(* CODESYS project EDS_V2_neu.project

Project tree, tasks and I/O mapping:
  CODESYS_SoftMotion_Win_V3 : CODESYS SoftMotion Win V3, 3S - Smart Software Solutions GmbH, order no. 309021, version 3.5.10.20
    application Application
      libraries: crane-control-lib, 1.0.3 (TUD)
      task VISU_TASK (cyclic, interval 100 ms, priority 31) calls VisuElems.Visu_Prg
      task Task (cyclic, interval t#20ms, priority 1) calls Motion_PRG_Motion, Motion_PRG_Control
      visualisation Visualization
      function block Bandsteuerung [SFC]: Init_active, Gleiten_active, Brems_active
      global variables GVL
      function Vmax [ST]
      program Motion_PRG_Control [FBD]
      program Motion_PRG_Motion [FBD]
      function block Kransteuerung [SFC]: brems_aufw_active, beschl_abw_active, Ruhelage_active
    SoftMotion General Axis Pool
      VA1_Band : SM_Drive_Virtual, 3S - Smart Software Solutions GmbH, order no. 1805, version 4.0.0.0
          settings: wDriveID = 0; iMovementType = 0
      VA2_Kran : SM_Drive_Virtual, 3S - Smart Software Solutions GmbH, order no. 1805, version 4.0.0.0
  libraries: VisuSymbols, 3.5.10.0 (System)
  text list GlobalTextList
*)

// CODESYS_SoftMotion_Win_V3/Application/GVL
VAR_GLOBAL
	
	jerk:REAL := 0; //unendlicher Ruck für geschwindigkeitsoptimale Steuerung
(* Steuervariablen (werden durch die Visualisierung gesetzt) *)
	Anlage_Ein:BOOL:=FALSE; (* Steuervariable zum Ein- und Ausschalten der Anlage *)
	Erzeuge_Paket_schwarz:BOOL; (* Es soll ein neues schwarzes Paket erzeugt werden *)
	Erzeuge_Paket_rot:BOOL; (* Es soll ein neues rotes Paket erzeugt werden *)
	
	(* Achsbezogene Variablen (repraesentieren aktuelle Messwerte der Achsen) *)
	Vact_Foerderbandachse:REAL; (* Aktuelle Winkelgeschwindigkeit der Foerderbandachse (in Grad/s) *)
	Vact_Foerderband:REAL; (* Aktuelle Geschwindigkeit des Foerderbandes (in mm/s) *)
	Vact_Kran1:REAL; (* Aktuelle vertikale Geschwindigkeit von Kran 1 (in mm/s) *)
	Posact_Kran1:REAL; (* Aktuelle vertikale Position von Kran 1 (in mm) *)
	
	(* Sensoren (werden durch den Simulator gesetzt) *)
	Messwert_Farbsensor:INT; (* Aktueller Messwert des Farbsensors (0=kein Paket; CONST.SCHWARZ=schwarzes Paket; CONST.ROT=rotes Paket) *)
	Kran1_In_Startpos:BOOL; (* Kran 1 befindet sich in seiner Startposition *)
	Kran1_In_Greifpos:BOOL; (* Kran 1 befindet sich in seiner Greifposition *)
	A_Band:REAL:=100;//*CONST.PI/180*RADIUS_FOERDERBANDACHSE; //Förderbeschleunigung Band in mm/s^2 //in Grad/s^2
	V_Band:REAL:=50;//*CONST.PI/180*RADIUS_FOERDERBANDACHSE ;//in mm/s //in Grad/s
	
	deltaT:REAL:=(GREIFPOS_X_KRAN1-POS_X_SENSOR)/(V_Band);(* berechnete Zeit des Paketes von Sensor zu Kran = Bewegungszeit des Krans in eine Richtung = 11.37s*)
	
END_VAR

// CODESYS_SoftMotion_Win_V3/Application/Motion_PRG_Motion
PROGRAM Motion_PRG_Motion
VAR_OUTPUT
	br_PowerVA1: BOOL;
	bd_PowerVA1: BOOL;
	bu_PowerVA1: BOOL;
	er_PowerVA1: BOOL;
	ID_PowerVA1: SMC_ERROR;
	st_PowerVA1: BOOL;
	
	don_accVA1: BOOL;
	bu_accVA1: BOOL;
	ab_accVA1: BOOL;
	er_accVA1: BOOL;
	ID_accVA1: SMC_ERROR;
	
	inVelocity_glVA1: BOOL;
	bu_glVA1: BOOL;
	ab_glVA1: BOOL;
	er_glVA1: BOOL;
	ID_glVA1: SMC_ERROR;
	
	don_decVA1: BOOL;
	bu_decVA1: BOOL;
	er_decVA1: BOOL;
	ID_decVA1: SMC_ERROR;
	
	
	st_PowerVA2: BOOL;
	bd_PowerVA2: BOOL;
	bu_PowerVA2: BOOL;
	br_PowerVA2: BOOL;
	er_PowerVA2: BOOL;
	ID_PowerVA2: SMC_ERROR;
	
	don_accVA2: BOOL;
	bu_accVA2: BOOL;
	er_accVA2: BOOL;
	ab_accVA2: BOOL;
	ID_accVA2: SMC_ERROR;
	
	inVelocity_glVA2: BOOL;
	bu_glVA2: BOOL;
	ab_glVA2: BOOL;
	ID_glVA2: SMC_ERROR;
	er_glVA2: BOOL;
	
	don_decVA2: BOOL;
	bu_decVA2: BOOL;
	er_decVA2: BOOL;
	ID_decVA2: SMC_ERROR;
	
END_VAR

VAR
	Power_VA1: MC_Power;
	Power_VA2: MC_Power;
	MC_Stop_Kran: MC_Stop;
	MC_MoveAbsolute_Kran: MC_MoveAbsolute;
	MC_MoveVelocity_Kran: MC_MoveVelocity;
	MC_MoveVelocity_Band :MC_MoveVelocity;
	MC_MoveAbsolute_Band: MC_MoveAbsolute;
	MC_Stop_Band: MC_Stop;
	
	
	
	don_reset: BOOL;
	bu_reset: BOOL;
	er_reset: BOOL;
	ID_reset: SMC_ERROR;
	MC_Reset_Band: MC_Reset;
	MC_Reset_Kran: MC_Reset;
END_VAR

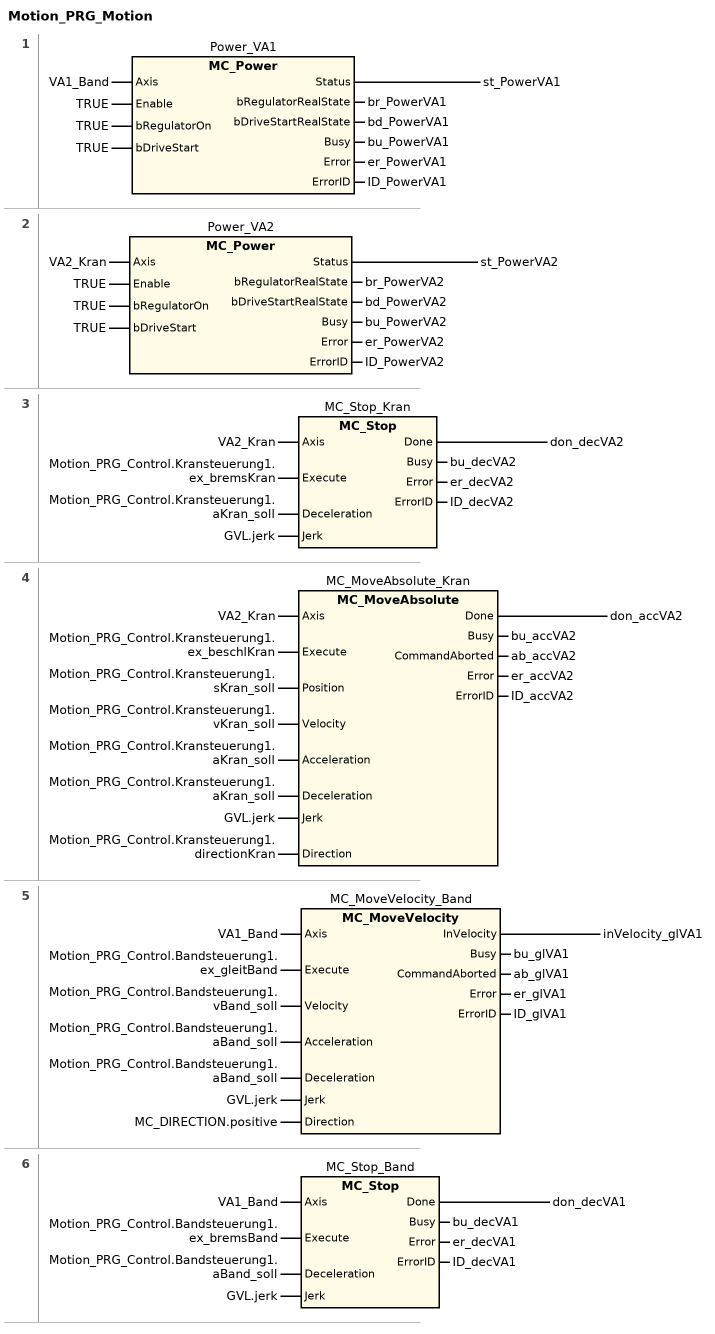
// NETWORK 1
Power_VA1(
    Axis := VA1_Band,
    Enable := TRUE,
    bRegulatorOn := TRUE,
    bDriveStart := TRUE,
    bRegulatorRealState => br_PowerVA1,
    bDriveStartRealState => bd_PowerVA1,
    Busy => bu_PowerVA1,
    Error => er_PowerVA1,
    ErrorID => ID_PowerVA1); // MC_Power
st_PowerVA1 := Power_VA1.Status;

// NETWORK 2
Power_VA2(
    Axis := VA2_Kran,
    Enable := TRUE,
    bRegulatorOn := TRUE,
    bDriveStart := TRUE,
    bRegulatorRealState => br_PowerVA2,
    bDriveStartRealState => bd_PowerVA2,
    Busy => bu_PowerVA2,
    Error => er_PowerVA2,
    ErrorID => ID_PowerVA2); // MC_Power
st_PowerVA2 := Power_VA2.Status;

// NETWORK 3
MC_Stop_Kran(
    Axis := VA2_Kran,
    Execute := Motion_PRG_Control.Kransteuerung1.ex_bremsKran,
    Deceleration := Motion_PRG_Control.Kransteuerung1.aKran_soll,
    Jerk := GVL.jerk,
    Busy => bu_decVA2,
    Error => er_decVA2,
    ErrorID => ID_decVA2); // MC_Stop
don_decVA2 := MC_Stop_Kran.Done;

// NETWORK 4
MC_MoveAbsolute_Kran(
    Axis := VA2_Kran,
    Execute := Motion_PRG_Control.Kransteuerung1.ex_beschlKran,
    Position := Motion_PRG_Control.Kransteuerung1.sKran_soll,
    Velocity := Motion_PRG_Control.Kransteuerung1.vKran_soll,
    Acceleration := Motion_PRG_Control.Kransteuerung1.aKran_soll,
    Deceleration := Motion_PRG_Control.Kransteuerung1.aKran_soll,
    Jerk := GVL.jerk,
    Direction := Motion_PRG_Control.Kransteuerung1.directionKran,
    Busy => bu_accVA2,
    CommandAborted => ab_accVA2,
    Error => er_accVA2,
    ErrorID => ID_accVA2); // MC_MoveAbsolute
don_accVA2 := MC_MoveAbsolute_Kran.Done;

// NETWORK 5
MC_MoveVelocity_Band(
    Axis := VA1_Band,
    Execute := Motion_PRG_Control.Bandsteuerung1.ex_gleitBand,
    Velocity := Motion_PRG_Control.Bandsteuerung1.vBand_soll,
    Acceleration := Motion_PRG_Control.Bandsteuerung1.aBand_soll,
    Deceleration := Motion_PRG_Control.Bandsteuerung1.aBand_soll,
    Jerk := GVL.jerk,
    Direction := MC_DIRECTION.positive,
    Busy => bu_glVA1,
    CommandAborted => ab_glVA1,
    Error => er_glVA1,
    ErrorID => ID_glVA1); // MC_MoveVelocity
inVelocity_glVA1 := MC_MoveVelocity_Band.InVelocity;

// NETWORK 6
MC_Stop_Band(
    Axis := VA1_Band,
    Execute := Motion_PRG_Control.Bandsteuerung1.ex_bremsBand,
    Deceleration := Motion_PRG_Control.Bandsteuerung1.aBand_soll,
    Jerk := GVL.jerk,
    Busy => bu_decVA1,
    Error => er_decVA1,
    ErrorID => ID_decVA1); // MC_Stop
don_decVA1 := MC_Stop_Band.Done;

END_PROGRAM

// CODESYS_SoftMotion_Win_V3/Application/Motion_PRG_Control
PROGRAM Motion_PRG_Control
VAR
	Simulator1:Simulator; (* Foerderbandsimulator aus der 'crane-control-lib' *)
	
	
	Kransteuerung1: Kransteuerung;
	Bandsteuerung1: Bandsteuerung;

	
	
END_VAR

VAR_OUTPUT
	
	ex_gleitBand: BOOL;
	ex_bremsBand: BOOL;
	ex_beschlKran: BOOL;
	ex_gleitKran: BOOL;
	ex_bremsKran:BOOL;
	aKran_soll:LREAL;
	vKran_soll:LREAL; //Sollwert der vertikalen Geschwindigkeit des Krans in mm/s
	sKran_soll:LREAL; //Sollwert des vertikalen Weges des Krans in mm 
	vBand_soll: LREAL;
	aBand_soll:LREAL;		
	ex_beschlBand: BOOL;
END_VAR

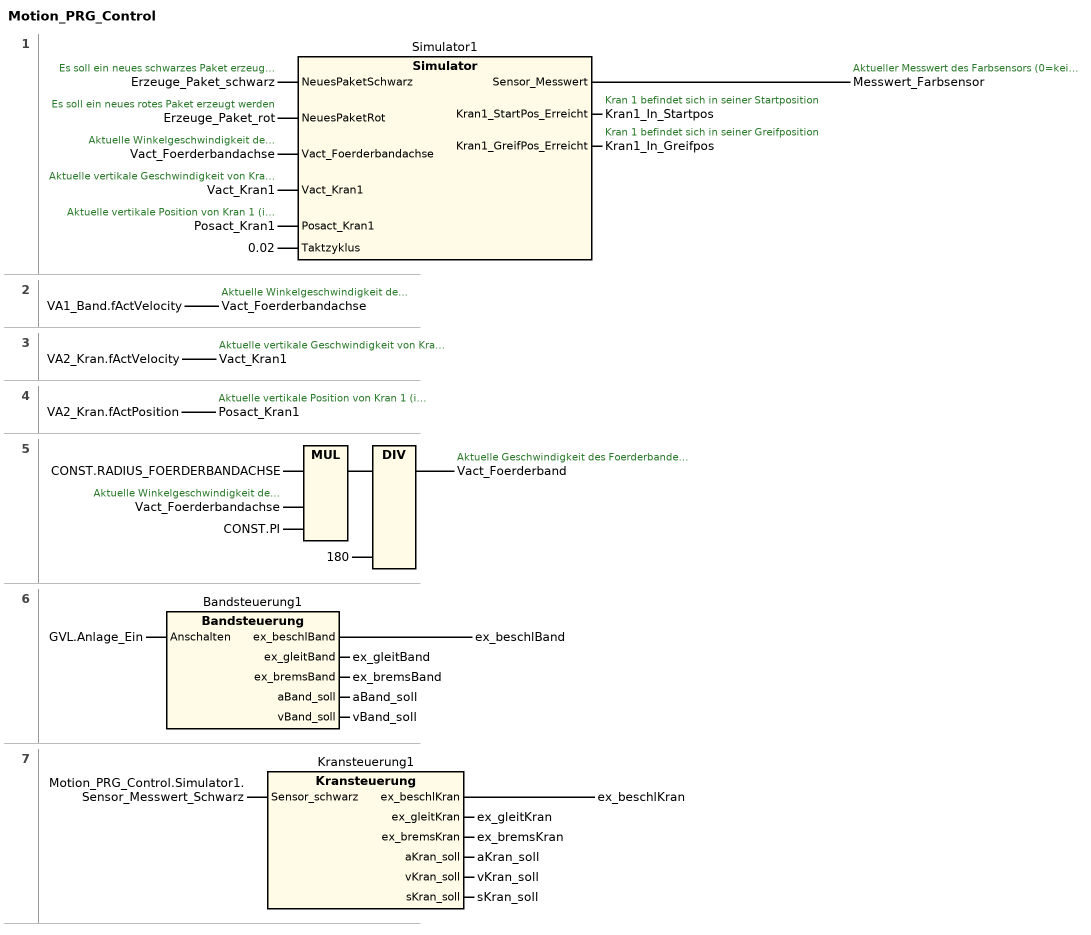
// NETWORK 1
//   Simulator1: Foerderbandsimulator aus der 'crane-control-lib'
//   Erzeuge_Paket_schwarz: Es soll ein neues schwarzes Paket erzeugt werden
//   Erzeuge_Paket_rot: Es soll ein neues rotes Paket erzeugt werden
//   Vact_Foerderbandachse: Aktuelle Winkelgeschwindigkeit der Foerderbandachse (in Grad/s)
//   Vact_Kran1: Aktuelle vertikale Geschwindigkeit von Kran 1 (in mm/s)
//   Posact_Kran1: Aktuelle vertikale Position von Kran 1 (in mm)
//   Kran1_In_Startpos: Kran 1 befindet sich in seiner Startposition
//   Kran1_In_Greifpos: Kran 1 befindet sich in seiner Greifposition
//   Messwert_Farbsensor: Aktueller Messwert des Farbsensors (0=kein Paket; CONST.SCHWARZ=schwarzes Paket; CONST.ROT=rotes Paket)
Simulator1(
    NeuesPaketSchwarz := Erzeuge_Paket_schwarz,
    NeuesPaketRot := Erzeuge_Paket_rot,
    Vact_Foerderbandachse := Vact_Foerderbandachse,
    Vact_Kran1 := Vact_Kran1,
    Posact_Kran1 := Posact_Kran1,
    Taktzyklus := 0.02,
    Kran1_StartPos_Erreicht => Kran1_In_Startpos,
    Kran1_GreifPos_Erreicht => Kran1_In_Greifpos); // Simulator
Messwert_Farbsensor := Simulator1.Sensor_Messwert;

// NETWORK 2
//   Vact_Foerderbandachse: Aktuelle Winkelgeschwindigkeit der Foerderbandachse (in Grad/s)
Vact_Foerderbandachse := VA1_Band.fActVelocity;

// NETWORK 3
//   Vact_Kran1: Aktuelle vertikale Geschwindigkeit von Kran 1 (in mm/s)
Vact_Kran1 := VA2_Kran.fActVelocity;

// NETWORK 4
//   Posact_Kran1: Aktuelle vertikale Position von Kran 1 (in mm)
Posact_Kran1 := VA2_Kran.fActPosition;

// NETWORK 5
//   Vact_Foerderbandachse: Aktuelle Winkelgeschwindigkeit der Foerderbandachse (in Grad/s)
//   Vact_Foerderband: Aktuelle Geschwindigkeit des Foerderbandes (in mm/s)
Vact_Foerderband := (CONST.RADIUS_FOERDERBANDACHSE * Vact_Foerderbandachse * CONST.PI) / 180;

// NETWORK 6
Bandsteuerung1(
    Anschalten := GVL.Anlage_Ein,
    ex_gleitBand => ex_gleitBand,
    ex_bremsBand => ex_bremsBand,
    aBand_soll => aBand_soll,
    vBand_soll => vBand_soll); // Bandsteuerung
ex_beschlBand := Bandsteuerung1.ex_beschlBand;

// NETWORK 7
Kransteuerung1(
    Sensor_schwarz := Motion_PRG_Control.Simulator1.Sensor_Messwert_Schwarz,
    ex_gleitKran => ex_gleitKran,
    ex_bremsKran => ex_bremsKran,
    aKran_soll => aKran_soll,
    vKran_soll => vKran_soll,
    sKran_soll => sKran_soll); // Kransteuerung
ex_beschlKran := Kransteuerung1.ex_beschlKran;

END_PROGRAM

// CODESYS_SoftMotion_Win_V3/Application/Bandsteuerung
FUNCTION_BLOCK Bandsteuerung


VAR
	TAU1 :TIME :=REAL_TO_TIME(V_Band/A_Band*10000);
	T1: BOOL:=FALSE;
	T2: BOOL:=FALSE;
END_VAR

VAR_OUTPUT
	ex_resetBand:BOOL:=FALSE;
	ex_beschlBand: BOOL:=FALSE;
	ex_gleitBand: BOOL:=FALSE;
	ex_bremsBand: BOOL:=FALSE;
	aBand_soll: LREAL;
	vBand_soll: LREAL;
	sBand_soll: LREAL;
END_VAR

VAR_INPUT
	Anschalten:BOOL:=GVL.Anlage_Ein;
END_VAR

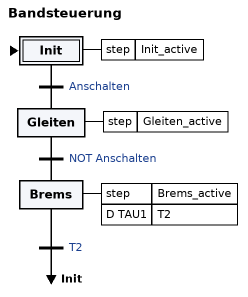
INITIAL_STEP Init:
    Init_active(N);  // step action
END_STEP
TRANSITION FROM Init TO Gleiten
    := Anschalten;
END_TRANSITION
STEP Gleiten:
    Gleiten_active(N);  // step action
END_STEP
TRANSITION FROM Gleiten TO Brems
    := NOT Anschalten;
END_TRANSITION
STEP Brems:
    Brems_active(N);  // step action
    T2(D, TAU1);
END_STEP
TRANSITION FROM Brems TO Init
    := T2;
END_TRANSITION

ACTION Init_active:

END_ACTION

ACTION Gleiten_active:
ex_beschlBand:=FALSE;
ex_gleitBand:=TRUE;
ex_bremsBand:=FALSE;
aBand_soll:=GVL.A_Band;
vBand_soll:=GVL.V_Band ;
END_ACTION

ACTION Brems_active:

ex_beschlBand:=FALSE;
ex_gleitBand:=FALSE;
ex_bremsBand:=TRUE;
aBand_soll:=A_Band;
vBand_soll:=0 ;
END_ACTION

END_FUNCTION_BLOCK

// CODESYS_SoftMotion_Win_V3/Application/Kransteuerung
FUNCTION_BLOCK Kransteuerung
VAR_INPUT
	Sensor_schwarz: BOOL := FALSE;
END_VAR

VAR_OUTPUT
	ex_resetKran:BOOL:=FALSE;
	directionKran:MC_DIRECTION;
	ex_beschlKran:BOOL;
	ex_gleitKran:BOOL;
	ex_bremsKran:BOOL;
	aKran_soll:LREAL;
	vKran_soll:LREAL; //Sollwert der vertikalen Geschwindigkeit des Krans in mm/s
	sKran_soll:LREAL; //Sollwert des vertikalen Weges des Krans in mm 
END_VAR

VAR
	deltaS:LREAL := CONST.GREIFPOS_Y_KRAN-CONST.STARTPOS_Y_KRAN;
	V_max:LREAL:= Vmax(deltaS,GVL.deltaT,CONST.A_MAX);
	TAU1:TIME := LREAL_TO_TIME(V_max/CONST.A_MAX*1000) ;
	TAU2:TIME := LREAL_TO_TIME((deltaS/V_max-V_max/CONST.A_MAX)*1000);
	TAU3:TIME := TAU1;
	t0: BOOL := FALSE;
	t1: BOOL := FALSE;
	t2: BOOL := FALSE;
	t3: BOOL := FALSE;
	t4: BOOL := FALSE;
	t5: BOOL := FALSE;
	t6: BOOL := FALSE;
	
	
	
END_VAR

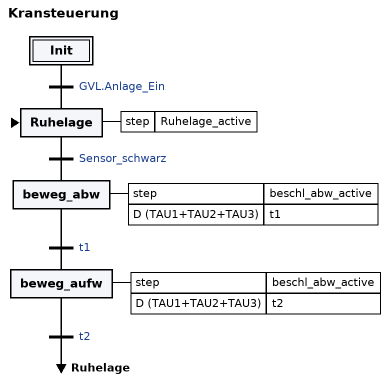
INITIAL_STEP Init:
END_STEP
TRANSITION FROM Init TO Ruhelage
    := GVL.Anlage_Ein;
END_TRANSITION
STEP Ruhelage:
    Ruhelage_active(N);  // step action
END_STEP
TRANSITION FROM Ruhelage TO beweg_abw
    := Sensor_schwarz;
END_TRANSITION
STEP beweg_abw:
    beschl_abw_active(N);  // step action
    t1(D, (TAU1+TAU2+TAU3));
END_STEP
TRANSITION FROM beweg_abw TO beweg_aufw
    := t1;
END_TRANSITION
STEP beweg_aufw:
    beschl_abw_active(N);  // step action
    t2(D, (TAU1+TAU2+TAU3));
END_STEP
TRANSITION FROM beweg_aufw TO Ruhelage
    := t2;
END_TRANSITION

ACTION brems_aufw_active:
ex_resetKran:=TRUE;
END_ACTION

ACTION beschl_abw_active:
ex_beschlKran:=TRUE;
ex_gleitKran:=FALSE;
ex_bremsKran:=FALSE;
aKran_soll:=CONST.A_MAX;
vKran_soll:=V_max;
sKran_soll:=CONST.STARTPOS_Y_KRAN;
directionKran:= MC_DIRECTION.negative;
END_ACTION

ACTION Ruhelage_active:
ex_beschlKran:=FALSE;
ex_gleitKran:=FALSE;
ex_bremsKran:=TRUE;

sKran_soll:=CONST.STARTPOS_Y_KRAN;
END_ACTION

END_FUNCTION_BLOCK

// CODESYS_SoftMotion_Win_V3/Application/Vmax
FUNCTION Vmax : LREAL
VAR_INPUT
	deltaS:LREAL;
	deltaT:LREAL;
	aMax:LREAL;
END_VAR
VAR
END_VAR

Vmax := deltaT*aMax/2*(1-SQRT(1-4*deltaS*aMax/EXPT(deltaT*aMax,2)));

END_FUNCTION

// CODESYS_SoftMotion_Win_V3/Application/Visualization
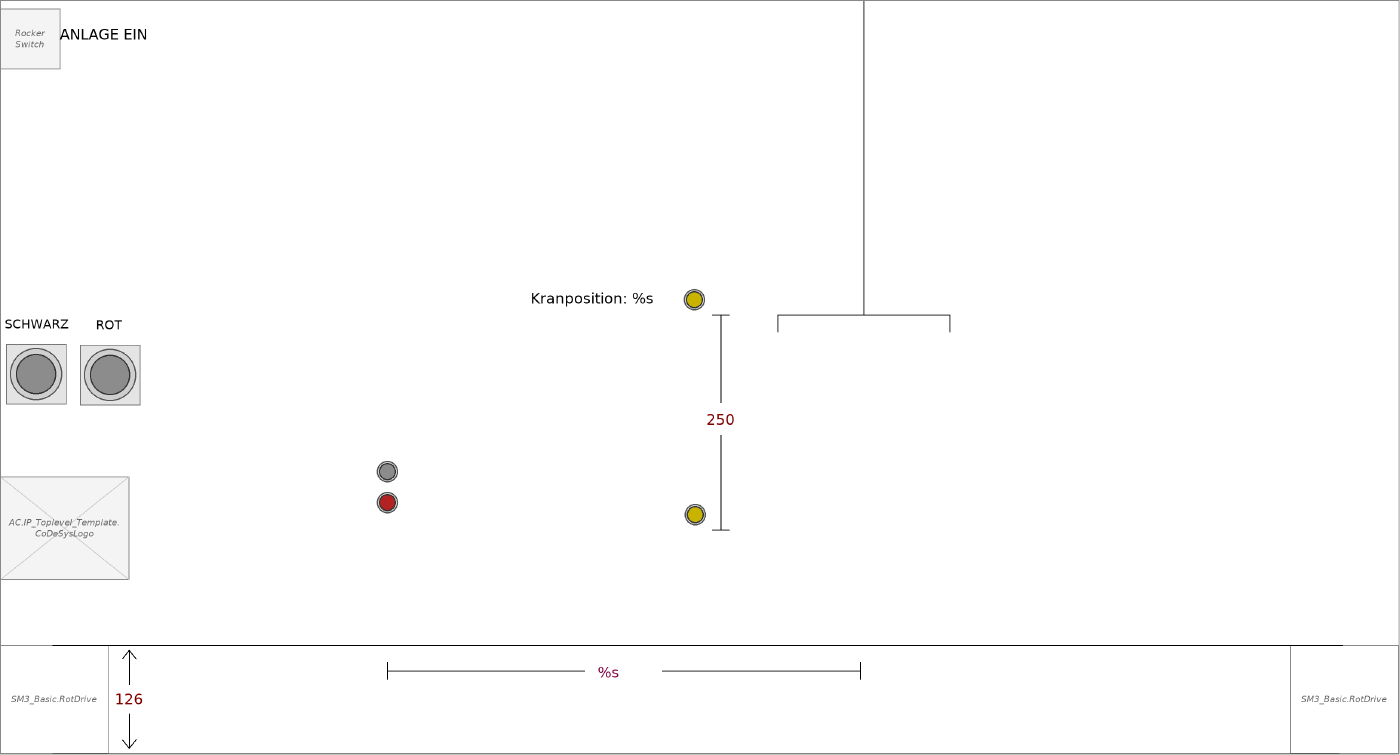
VISUALIZATION Visualization  // 1628x878
    Group (615,-2 490x619)
        p3560616238: GREIFPOS_X_KRAN1-925
        Line (389,0) (389,360)
        Line (389,50) (389,368)
            p2738717112: VA2_Kran.fActPosition
        Line (289,368) (489,368)
            p2738717112: VA2_Kran.fActPosition
        Line (489,368) (489,388)
            p2738717112: VA2_Kran.fActPosition
        Line (289,368) (289,388)
            p2738717112: VA2_Kran.fActPosition
        Textfield (117,334 60x30), "%s", text variable: Posact_Kran1
        Lamp1 (178,586 31x29), variable: Motion_PRG_Control.Simulator1.Kran1_GreifPos_Erreicht, style: Lamp-Lamp1-Yellow
        Lamp1 (177,336 31x29), variable: Motion_PRG_Control.Simulator1.Kran1_StartPos_Erreicht, style: Lamp-Lamp1-Yellow
        Line (223,368) (223,470)
        Line (223,508) (223,618)
        Label (189,473 68x34), "250"
        Line (213,618) (233,618)
        Line (213,368) (233,368)
        Label (0,334 117x30), "Kranposition:"
    Frame (0,750 126x126)
        shows SM3_Basic.RotDrive(m_Input_AXISREF := VA1_Band)
    Frame (1500,750 126x126)
        shows SM3_Basic.RotDrive(m_Input_AXISREF := VA1_Band)
        p3560616238: LAENGE_FOERDERBAND-1500
    Line (0,0) (1626,0)
    RockerSwitch (0,10 70x70), variable: GVL.Anlage_Ein, behaviour: TOGGLE, style: Switch-RockerSwitch-Gray
    Image (0,554 150x120), colour toggle: INT_TO_BOOL(Motion_PRG_Control.Simulator1.Paket1_Farbe - 1), invisible if: Motion_PRG_Control.Simulator1.Paket1_Unsichtbar, image: AC.IP_Toplevel_Template.CoDeSysLogo
        p3560616238: Motion_PRG_Control.Simulator1.Paket1_Pos_x
        p2738717112: Motion_PRG_Control.Simulator1.Paket1_Pos_y
    PushSwitch (7,400 70x70), variable: Erzeuge_Paket_schwarz, behaviour: TAP, style: Switch-PushSwitch-Gray
    Image (0,554 150x120), colour toggle: INT_TO_BOOL(Motion_PRG_Control.Simulator1.Paket2_Farbe - 1), invisible if: Motion_PRG_Control.Simulator1.Paket2_Unsichtbar, image: AC.IP_Toplevel_Template.CoDeSysLogo
        p3560616238: Motion_PRG_Control.Simulator1.Paket2_Pos_x
        p2738717112: Motion_PRG_Control.Simulator1.Paket2_Pos_y
    Line (61,750) (1061,750)
    Line (61,876) (1061,876)
    Label (0,360 86x34), "SCHWARZ"
    Label (56,23 129x34), "ANLAGE EIN"
    Lamp1 (435,534 31x29), variable: Motion_PRG_Control.Simulator1.Sensor_Messwert_Schwarz, style: Lamp-Lamp1-Gray
    Line (450,780) (650,780)
    Line (450,770) (450,790)
    Line (1000,770) (1000,790)
        p3560616238: GREIFPOS_X_KRAN1-925
    Line (770,780) (970,780)
        p3560616238: (GREIFPOS_X_KRAN1-925)/2
    Line (364,317)
    Line (150,756) (150,796)
    Line (150,830) (150,870)
    Label (116,796 68x34), "126"
    Line (150,756) (158,766)
    Line (150,756) (142,766)
    Line (142,860) (150,870)
    Line (158,860) (150,870)
    Line (561,750) (1561,750)
        p3560616238: LAENGE_FOERDERBAND-1500
    Line (557,876) (1557,876)
        p3560616238: LAENGE_FOERDERBAND-1500
    Line (480,780) (680,780)
        p3560616238: (GREIFPOS_X_KRAN1-925)/2
    Line (800,780) (1000,780)
        p3560616238: (GREIFPOS_X_KRAN1-925)/2
    Textfield (692,765 68x34), "%s", text variable: CONST.GREIFPOS_X_KRAN1 - CONST.POS_X_SENSOR
    Lamp1 (435,570 31x29), variable: Motion_PRG_Control.Simulator1.Sensor_Messwert_Rot, style: Lamp-Lamp1-Red
    PushSwitch (93,401 70x70), variable: Erzeuge_Paket_rot, behaviour: TAP, style: Switch-PushSwitch-Gray
    Label (93,361 68x34), "ROT"
END_VISUALIZATION
